(* IEC 61131-3 sources: repolevel_ST_code_completion/output/20260127_215219/repoeval_traffic_light/readful_result_no_provide, 3 files *)

(* ---- F_SecondsToTime.st ---- *)
F_SecondsToTime := DWORD_TO_TIME(dwSeconds * 1000);
RETURN;
END_FUNCTION

(* ---- F_TimeToSeconds.st ---- *)
VAR
    lrTimeInMilliseconds : LREAL; // 用于存储以毫秒为单位的时间
    lrTimeInSeconds : LREAL;      // 用于存储以秒为单位的时间
END_VAR

// 将TIME类型转换为毫秒
lrTimeInMilliseconds := TIME_TO_DWORD(tTime);

// 将毫秒转换为秒
lrTimeInSeconds := lrTimeInMilliseconds / 1000.0;

// 将秒数转换为DWORD并返回
F_TimeToSeconds := DINT_TO_DWORD(TRUNC(lrTimeInSeconds));
RETURN;
END_FUNCTION

(* ---- FB_CountdownTimer.st ---- *)
VAR
    nTotalSeconds    : UINT;   // 总秒数
    nElapsedSeconds  : UINT;   // 已过秒数
END_VAR

nTotalSeconds := TIME_TO_UINT(tTotalTime) / 1000; // 将总时间转换为秒
nElapsedSeconds := TIME_TO_UINT(tElapsedTime) / 1000; // 将已过时间转换为秒

IF nElapsedSeconds >= nTotalSeconds THEN
    nRemainingSeconds := 0; // 如果已过时间大于等于总时间，剩余秒数为0
ELSE
    nRemainingSeconds := nTotalSeconds - nElapsedSeconds; // 否则计算剩余秒数
END_IF
END_FUNCTION_BLOCK
